FUNCTION_BLOCK FB_NTCLE_MOTOR
VAR_INPUT
	icriticalindex:		SINT := -1;
END_VAR
VAR_OUTPUT
	i:					USINT;
	TEMP: ARRAY[0..8] OF REAL;
	bcriticalCoolDown:			BOOL := FALSE;

	
END_VAR

VAR
	
	temp_raw11 AT %I*	:INT;
	temp_raw12 AT %I*	:INT;
	temp_raw13 AT %I*	:INT;
	temp_raw14 AT %I*	:INT;
	temp_raw15 AT %I*	:INT;
	temp_raw16 AT %I*	:INT;
	temp_raw17 AT %I*	:INT;
	temp_raw18 AT %I*	:INT;
	temp_raw19 AT %I*	:INT;
	
	
END_VAR

bcriticalCoolDown := FALSE;
icriticalindex := -1;

TEMP[0] := INT_TO_REAL(temp_raw11)/100.0;
TEMP[1] := INT_TO_REAL(temp_raw12)/100.0;
TEMP[2] := INT_TO_REAL(temp_raw13)/100.0;
TEMP[3] := INT_TO_REAL(temp_raw14)/100.0;
TEMP[4] := INT_TO_REAL(temp_raw15)/100.0;
TEMP[5] := INT_TO_REAL(temp_raw16)/100.0;
TEMP[6] := INT_TO_REAL(temp_raw17)/100.0;
TEMP[7] := INT_TO_REAL(temp_raw18)/100.0;
TEMP[8] := INT_TO_REAL(temp_raw19)/100.0;

FOR i := 0 TO 8 DO
	IF TEMP[i] > GVL_FSM.rcritical_temp_prop THEN
		
		GVL_THERMAL.bMOTOROVERHEAT := TRUE;
		icriticalindex := i;
		GVL_PROP.propulsion_fault := TRUE;
		
	END_IF
	IF TEMP[i] < GVL_FSM.rcritical_temp_prop_coolDown THEN
		
		bcriticalCoolDown := TRUE;
		
	END_IF
END_FOR
IF icriticalindex <> -1 THEN
	bcriticalCoolDown := FALSE;
END_IF

END_FUNCTION_BLOCK

(* stored: Version 1.1.0.1
   POU FB_NTCLE_MOTOR: Id {016e6a52-5f4e-431c-a5b7-741f994aab92}, SpecialFunc None *)
